Omron CX-Programmer project NewProject (CX-Programmer 9.73)

# PLC NewPLC1: CP2E-N N

## Global symbols (name address type ; comment)
0.00 BOOL  ; PB_EMG
0.01 BOOL  ; Sensor 1m
0.02 BOOL  ; Sensor 1,5 M
0.04 BOOL  ; Sensor Drop
0.06 BOOL  ; Sensor Clean BWD
0.07 BOOL  ; S Home 2
0.08 BOOL  ; S Home 2
0.11 BOOL  ; EMG/PB
100.04 BOOL  ; Q_Break1
100.05 BOOL  ; Q_Break2
100.06 BOOL  ; Q_EN1
100.07 BOOL  ; Q_EN2
101.00 BOOL  ; Cylinder_CLEAN
101.01 BOOL  ; Cylinder_DROP
101.02 BOOL  ; Motor_Down
101.03 BOOL  ; Motor_Up
101.07 BOOL  ; Test Break
200 CHANNEL  ; Timer Clean
280.07 BOOL  ; Ax0 Error
A274 CHANNEL  ; Ax1 Pulse
A276 CHANNEL  ; Ax0 Current PLS
A277 CHANNEL  ; Ax1 Current PLS
A278 CHANNEL  ; Ax1 Pulse Org
A280.04 BOOL  ; Ax0 Busy
A280.05 BOOL  ; Ax0 No Org
A280.06 BOOL  ; Ax0 at Org
A280.07 BOOL  ; Ax0 Error
A281.04 BOOL  ; Ax1 Bussy
A286 CHANNEL  ; Ax1 Current PLS
A540.08 BOOL  ; Ax0 CW-Limit Input
A540.09 BOOL  ; Ax0 CCW-Limit Input
D0 CHANNEL  ; $?St$Bk?_#[4] / Value"0"$?St$Bk?_#[4]
D10 CHANNEL  ; Point A Data
D100 CHANNEL  ; Axo Acceleration
D101 CHANNEL  ; Ax0 Deceleration
D102 CHANNEL  ; Target Frequency
D104 CHANNEL  ; Ax0 Number PLS Output
D105 CHANNEL  ; Ax1 Number PLS Output
D106 CHANNEL  ; Start Frequency
D110 CHANNEL  ; Ax1 Acceleration
D111 CHANNEL  ; Ax1 Deceleration
D112 CHANNEL  ; Target Frequency1
D114 CHANNEL  ; Ax1 Number PLS Output
D116 CHANNEL  ; Start Frequncy1
D12 CHANNEL  ; Point B Data
D120 CHANNEL  ; Ax1 Acceleration
D124 CHANNEL  ; Ax1 Number PLS Output
D126 CHANNEL  ; Start Frequency
D14 CHANNEL  ; Point C Data
D20 CHANNEL  ; Point A2 Data
D22 CHANNEL  ; Point B2 Data
D24 CHANNEL  ; Point C2 Data
D276 CHANNEL  ; Ax0 Current PLS
D277 CHANNEL  ; Ax1 Current PLS
D278 CHANNEL  ; Ax1 PLS
D286 CHANNEL  ; Ax1 Current PLS
T002 BOOL  ; T Clean
T003 BOOL  ; Active DROP
T004 BOOL  ; Active Motor Up
T005 BOOL  ; Timer Continue
T010 BOOL  ; Ax0 Jog High
T011 BOOL  ; Ax1 Jog High
W0.02 BOOL  ; PB Ax0 Org
W0.03 BOOL  ; Axis0 Jog(+)
W0.04 BOOL  ; Axis Jog(-)
W0.05 BOOL  ; PB Ax1 Org
W0.06 BOOL  ; Axis1 Jog(+)
W0.07 BOOL  ; Axis1 Jog(-)
W0.08 BOOL  ; Init Done
W100.00 BOOL  ; No Use
W100.01 BOOL  ; BREAK ACTIVE
W100.02 BOOL  ; ENA 1
W100.03 BOOL  ; INI MOTOR
W100.04 BOOL  ; BREAK 2
W100.07 BOOL  ; ENA 2
W10.00 BOOL  ; Ax0 Recover Org Start
W10.01 BOOL  ; Ax0 Recover Org Start PLS
W10.02 BOOL  ; Ax0 Org Return
W10.03 BOOL  ; Ax0 Org Returning
W10.04 BOOL  ; Ax0 at Org
W10.05 BOOL  ; Init
W10.06 BOOL  ; Ax0 Moving
W10.14 BOOL  ; Ax1 Recover
W10.15 BOOL  ; Ax0 Recover C
W11.00 BOOL  ; 10.01
W11.01 BOOL  ; Ax1 Recover Org Start PLS
W11.10 BOOL  ; Teach A2
W11.11 BOOL  ; Teach B2
W11.12 BOOL  ; Teach C2
W12.00 BOOL  ; Button Home
W12.01 BOOL  ; M_Home 1
W12.02 BOOL  ; Sens Home 1
W12.03 BOOL  ; M_Break 1
W12.04 BOOL  ; M_Break 2
W12.10 BOOL  ; M1_Ready
W12.11 BOOL  ; M2_Ready
W12.12 BOOL  ; Break M1 Deactive
W12.13 BOOL  ; M2_Break Deactive
W13.00 BOOL  ; Button Home2
W13.01 BOOL  ; M_Home 2
W13.02 BOOL  ; Sens_Home2
W14.00 BOOL  ; Teach A2
W14.01 BOOL  ; Teach B2
W14.02 BOOL  ; Teach C2
W15.00 BOOL  ; Point A2 Run
W15.01 BOOL  ; Point B2 Run
W15.02 BOOL  ; Point C2 Run
W15.03 BOOL  ; Home All
W16.00 BOOL  ; IO Clean
W16.01 BOOL  ; IO DROP
W16.02 BOOL  ; M_Mtr_Down
W16.03 BOOL  ; UP 1.5m
W16.04 BOOL  ; Up 1m
W16.05 BOOL  ; FINISH
W16.06 BOOL  ; Go Up
W16.07 BOOL  ; Stop Home
W17.00 BOOL  ; Manual UP
W17.01 BOOL  ; Manual Down
W1.00 BOOL  ; Ax0 Jog High Speed
W1.01 BOOL  ; Ax0 Jog(+)
W1.02 BOOL  ; Ax0 Jog(-)
W1.03 BOOL  ; Ax1 Jog High Speed
W1.04 BOOL  ; Ax1 Jog(+)
W1.05 BOOL  ; Ax1 Jog(-)
W1.08 BOOL  ; Init Done2
W1.10 BOOL  ; Teach Point A
W1.11 BOOL  ; Teah Point B
W1.12 BOOL  ; Teach Point C
W20.00 BOOL  ; No Use
W20.01 BOOL  ; Sens Home
W20.02 BOOL  ; Sens CW
W20.03 BOOL  ; Sens CCW
W2.00 BOOL  ; Point A Run
W2.01 BOOL  ; Point B Run
W2.02 BOOL  ; Point C Run
W2.10 BOOL  ; Point A2 Run
W2.11 BOOL  ; Point B2 Run
W2.12 BOOL  ; Point C2 Run
W3.00 BOOL  ; Point A Proses
W3.01 BOOL  ; Point A Trigger
W3.02 BOOL  ; Ax0 at Point A
W3.10 BOOL  ; Point A2 Proses
W3.11 BOOL  ; Point A2 Trigger
W3.12 BOOL  ; Ax0 at Point A2
W4.00 BOOL  ; Point B Process
W4.01 BOOL  ; Point B Trigger
W4.02 BOOL  ; Ax0 at Point B
W4.10 BOOL  ; Point B2 Progress
W4.11 BOOL  ; Point B2 Trigger
W4.12 BOOL  ; Ax1 at Point B
W5.00 BOOL  ; Point C Progress
W5.01 BOOL  ; Point C Trigger
W5.02 BOOL  ; Ax0 at Point C
W5.10 BOOL  ; Point C2 Progress
W5.11 BOOL  ; Point C2 Trigger
W5.12 BOOL  ; Ax1 at Point C
W6.00 BOOL  ; Sensor Trig
W6.01 BOOL  ; Trig Off
W7.00 BOOL  ; PB_START
W7.01 BOOL  ; M_Start
W7.02 BOOL  ; PB_STOP
W7.03 BOOL  ; PB_HOME
W7.04 BOOL  ; RUN 1or1.5
W7.05 BOOL  ; RUN 1m
W7.06 BOOL  ; PB_Continue
W99.01 BOOL  ; LOCK

## Program NewProgram1 (cyclic task 0)
Local symbols
NOT BOOL

### Section Axis1_Org

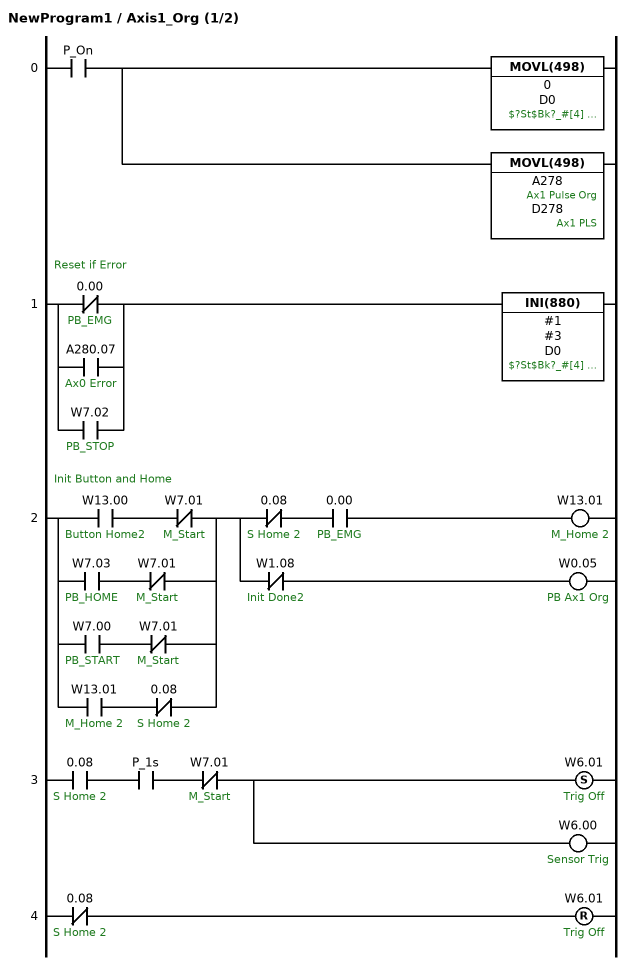
; rung 0
LD P_On
MOVL(498) 0 D0  ; $?St$Bk?_#[4] / Value"0"$?St$Bk?_#[4]
MOVL(498) A278 D278  ; Ax1 Pulse Org, Ax1 PLS
; rung 1: Reset if Error
LDNOT 0.00  ; PB_EMG
OR A280.07  ; Ax0 Error
OR W7.02  ; PB_STOP
INI(880) #1 #3 D0  ; $?St$Bk?_#[4] / Value"0"$?St$Bk?_#[4]
; rung 2: Init Button and Home
LD W13.00  ; Button Home2
ANDNOT W7.01  ; M_Start
LD W7.03  ; PB_HOME
ANDNOT W7.01  ; M_Start
ORLD
LD W7.00  ; PB_START
ANDNOT W7.01  ; M_Start
ORLD
LD W13.01  ; M_Home 2
ANDNOT 0.08  ; S Home 2
ORLD
OUT TR0
ANDNOT 0.08  ; S Home 2
AND 0.00  ; PB_EMG
OUT W13.01  ; M_Home 2
LD TR0
ANDNOT W1.08  ; Init Done2
OUT W0.05  ; PB Ax1 Org
; rung 3
LD 0.08  ; S Home 2
AND P_1s
ANDNOT W7.01  ; M_Start
SET W6.01  ; Trig Off
OUT W6.00  ; Sensor Trig
; rung 4
LDNOT 0.08  ; S Home 2
RSET W6.01  ; Trig Off

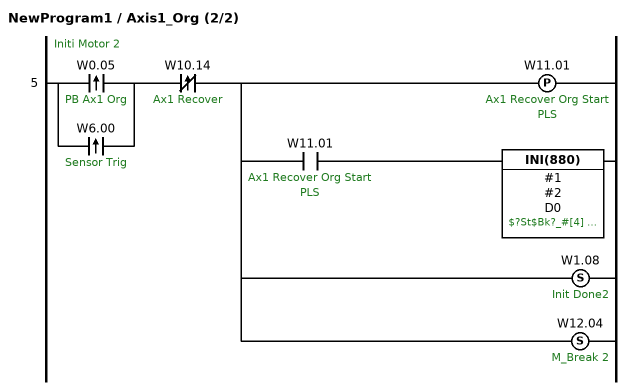
; rung 5: Initi Motor 2
@LD W0.05  ; PB Ax1 Org
@OR W6.00  ; Sensor Trig
@ANDNOT W10.14  ; Ax1 Recover
OUT TR0
DIFU(013) W11.01  ; Ax1 Recover Org Start PLS
AND W11.01  ; Ax1 Recover Org Start PLS
INI(880) #1 #2 D0  ; $?St$Bk?_#[4] / Value"0"$?St$Bk?_#[4]
LD TR0
SET W1.08  ; Init Done2
SET W12.04  ; M_Break 2

### Section Axis1_Jog

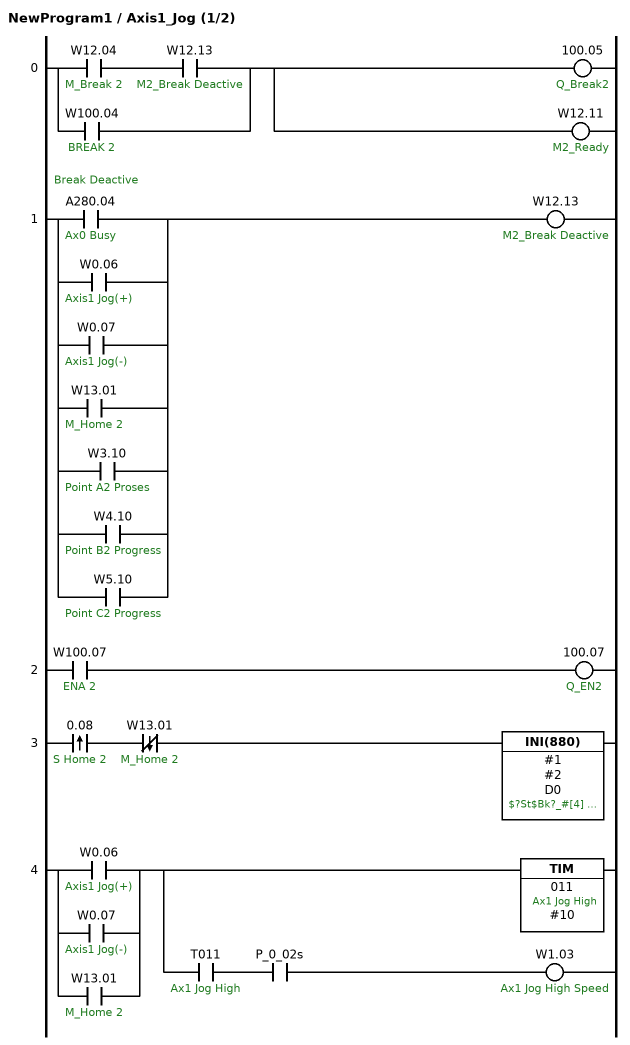
; rung 0
LD W12.04  ; M_Break 2
AND W12.13  ; M2_Break Deactive
OR W100.04  ; BREAK 2
OUT 100.05  ; Q_Break2
OUT W12.11  ; M2_Ready
; rung 1: Break Deactive
LD A280.04  ; Ax0 Busy
OR W0.06  ; Axis1 Jog(+)
OR W0.07  ; Axis1 Jog(-)
OR W13.01  ; M_Home 2
OR W3.10  ; Point A2 Proses
OR W4.10  ; Point B2 Progress
OR W5.10  ; Point C2 Progress
OUT W12.13  ; M2_Break Deactive
; rung 2
LD W100.07  ; ENA 2
OUT 100.07  ; Q_EN2
; rung 3
@LD 0.08  ; S Home 2
%ANDNOT W13.01  ; M_Home 2
INI(880) #1 #2 D0  ; $?St$Bk?_#[4] / Value"0"$?St$Bk?_#[4]
; rung 4
LD W0.06  ; Axis1 Jog(+)
OR W0.07  ; Axis1 Jog(-)
OR W13.01  ; M_Home 2
TIM 011 #10  ; Ax1 Jog High
AND T011  ; Ax1 Jog High
AND P_0_02s
OUT W1.03  ; Ax1 Jog High Speed

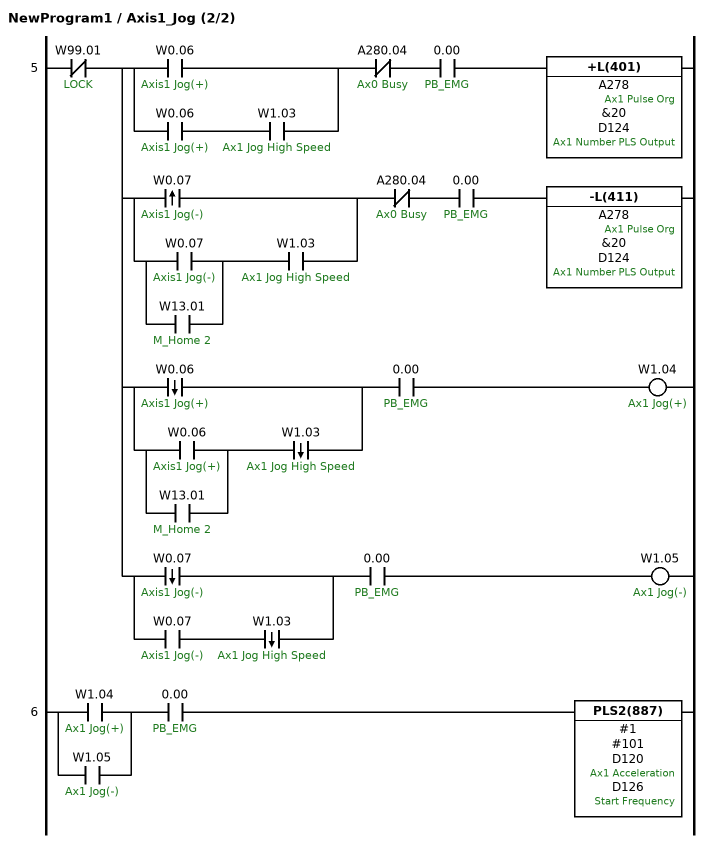
; rung 5
LDNOT W99.01  ; LOCK
OUT TR0
LD W0.06  ; Axis1 Jog(+)
LD W0.06  ; Axis1 Jog(+)
AND W1.03  ; Ax1 Jog High Speed
ORLD
ANDLD
ANDNOT A280.04  ; Ax0 Busy
AND 0.00  ; PB_EMG
+L(401) A278 &20 D124  ; Ax1 Pulse Org, Ax1 Number PLS Output
LD TR0
@LD W0.07  ; Axis1 Jog(-)
LD W0.07  ; Axis1 Jog(-)
OR W13.01  ; M_Home 2
AND W1.03  ; Ax1 Jog High Speed
ORLD
ANDLD
ANDNOT A280.04  ; Ax0 Busy
AND 0.00  ; PB_EMG
-L(411) A278 &20 D124  ; Ax1 Pulse Org, Ax1 Number PLS Output
LD TR0
%LD W0.06  ; Axis1 Jog(+)
LD W0.06  ; Axis1 Jog(+)
OR W13.01  ; M_Home 2
%AND W1.03  ; Ax1 Jog High Speed
ORLD
ANDLD
AND 0.00  ; PB_EMG
OUT W1.04  ; Ax1 Jog(+)
LD TR0
%LD W0.07  ; Axis1 Jog(-)
LD W0.07  ; Axis1 Jog(-)
%AND W1.03  ; Ax1 Jog High Speed
ORLD
ANDLD
AND 0.00  ; PB_EMG
OUT W1.05  ; Ax1 Jog(-)
; rung 6
LD W1.04  ; Ax1 Jog(+)
OR W1.05  ; Ax1 Jog(-)
AND 0.00  ; PB_EMG
PLS2(887) #1 #101 D120 D126  ; Ax1 Acceleration, Start Frequency

### Section Axis1_Point_Run

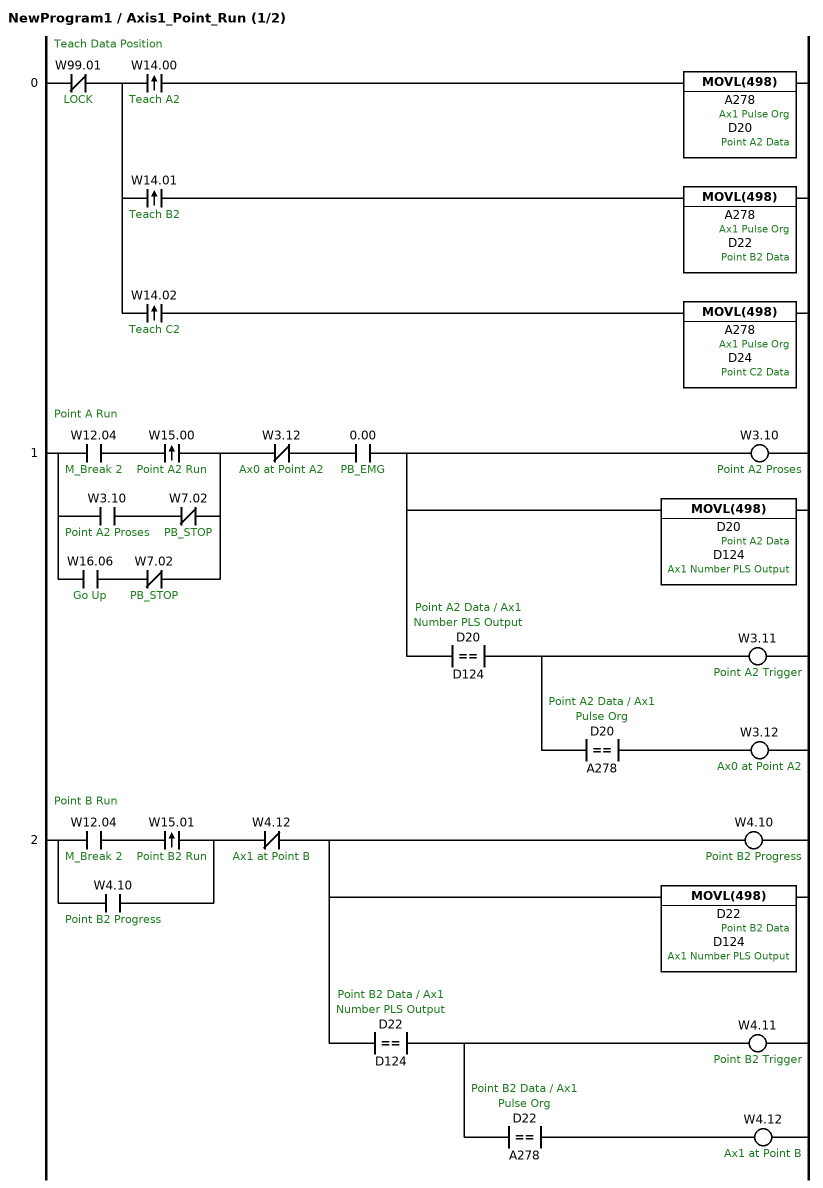
; rung 0: Teach Data Position
LDNOT W99.01  ; LOCK
OUT TR0
@AND W14.00  ; Teach A2
MOVL(498) A278 D20  ; Ax1 Pulse Org, Point A2 Data
LD TR0
@AND W14.01  ; Teach B2
MOVL(498) A278 D22  ; Ax1 Pulse Org, Point B2 Data
LD TR0
@AND W14.02  ; Teach C2
MOVL(498) A278 D24  ; Ax1 Pulse Org, Point C2 Data
; rung 1: Point A Run
LD W12.04  ; M_Break 2
@AND W15.00  ; Point A2 Run
LD W3.10  ; Point A2 Proses
ANDNOT W7.02  ; PB_STOP
ORLD
LD W16.06  ; Go Up
ANDNOT W7.02  ; PB_STOP
ORLD
ANDNOT W3.12  ; Ax0 at Point A2
AND 0.00  ; PB_EMG
OUT W3.10  ; Point A2 Proses
MOVL(498) D20 D124  ; Point A2 Data, Ax1 Number PLS Output
AND=L(301) D20 D124  ; Point A2 Data, Ax1 Number PLS Output
OUT W3.11  ; Point A2 Trigger
AND=L(301) D20 A278  ; Point A2 Data, Ax1 Pulse Org
OUT W3.12  ; Ax0 at Point A2
; rung 2: Point B Run
LD W12.04  ; M_Break 2
@AND W15.01  ; Point B2 Run
OR W4.10  ; Point B2 Progress
ANDNOT W4.12  ; Ax1 at Point B
OUT W4.10  ; Point B2 Progress
MOVL(498) D22 D124  ; Point B2 Data, Ax1 Number PLS Output
AND=L(301) D22 D124  ; Point B2 Data, Ax1 Number PLS Output
OUT W4.11  ; Point B2 Trigger
AND=L(301) D22 A278  ; Point B2 Data, Ax1 Pulse Org
OUT W4.12  ; Ax1 at Point B

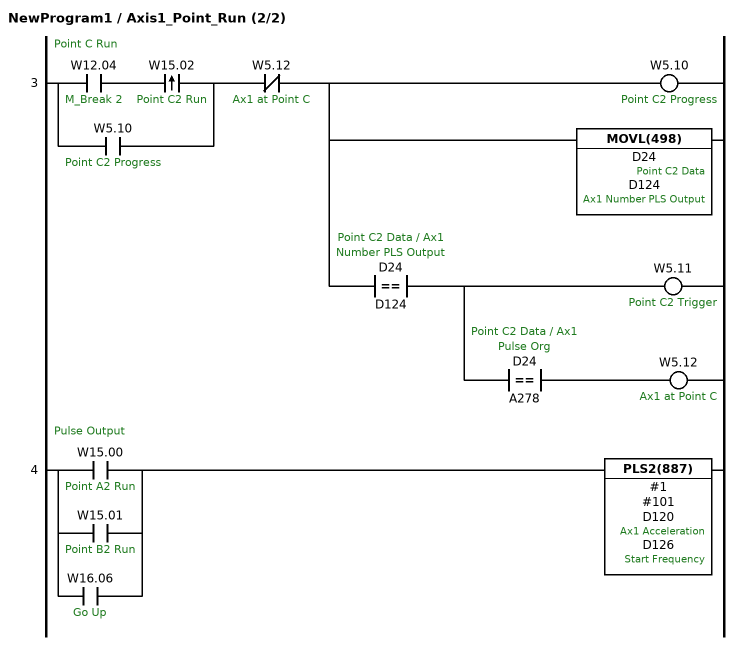
; rung 3: Point C Run
LD W12.04  ; M_Break 2
@AND W15.02  ; Point C2 Run
OR W5.10  ; Point C2 Progress
ANDNOT W5.12  ; Ax1 at Point C
OUT W5.10  ; Point C2 Progress
MOVL(498) D24 D124  ; Point C2 Data, Ax1 Number PLS Output
AND=L(301) D24 D124  ; Point C2 Data, Ax1 Number PLS Output
OUT W5.11  ; Point C2 Trigger
AND=L(301) D24 A278  ; Point C2 Data, Ax1 Pulse Org
OUT W5.12  ; Ax1 at Point C
; rung 4: Pulse Output
LD W15.00  ; Point A2 Run
OR W15.01  ; Point B2 Run
OR W16.06  ; Go Up
PLS2(887) #1 #101 D120 D126  ; Ax1 Acceleration, Start Frequency

### Section MOTOR_DROP_TEST

### Section Program

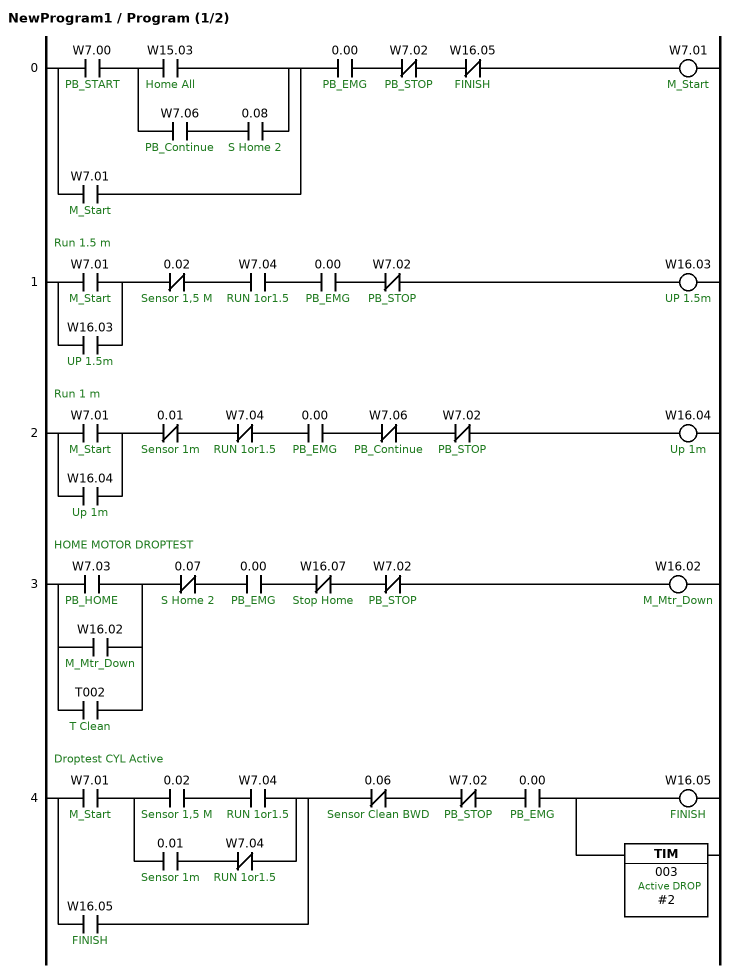
; rung 0
LD W7.00  ; PB_START
LD W15.03  ; Home All
LD W7.06  ; PB_Continue
AND 0.08  ; S Home 2
ORLD
ANDLD
OR W7.01  ; M_Start
AND 0.00  ; PB_EMG
ANDNOT W7.02  ; PB_STOP
ANDNOT W16.05  ; FINISH
OUT W7.01  ; M_Start
; rung 1: Run 1.5 m
LD W7.01  ; M_Start
OR W16.03  ; UP 1.5m
ANDNOT 0.02  ; Sensor 1,5 M
AND W7.04  ; RUN 1or1.5
AND 0.00  ; PB_EMG
ANDNOT W7.02  ; PB_STOP
OUT W16.03  ; UP 1.5m
; rung 2: Run 1 m
LD W7.01  ; M_Start
OR W16.04  ; Up 1m
ANDNOT 0.01  ; Sensor 1m
ANDNOT W7.04  ; RUN 1or1.5
AND 0.00  ; PB_EMG
ANDNOT W7.06  ; PB_Continue
ANDNOT W7.02  ; PB_STOP
OUT W16.04  ; Up 1m
; rung 3: HOME MOTOR DROPTEST
LD W7.03  ; PB_HOME
OR W16.02  ; M_Mtr_Down
OR T002  ; T Clean
ANDNOT 0.07  ; S Home 2
AND 0.00  ; PB_EMG
ANDNOT W16.07  ; Stop Home
ANDNOT W7.02  ; PB_STOP
OUT W16.02  ; M_Mtr_Down
; rung 4: Droptest CYL Active
LD W7.01  ; M_Start
LD 0.02  ; Sensor 1,5 M
AND W7.04  ; RUN 1or1.5
LD 0.01  ; Sensor 1m
ANDNOT W7.04  ; RUN 1or1.5
ORLD
ANDLD
OR W16.05  ; FINISH
ANDNOT 0.06  ; Sensor Clean BWD
ANDNOT W7.02  ; PB_STOP
AND 0.00  ; PB_EMG
OUT W16.05  ; FINISH
TIM 003 #2  ; Active DROP

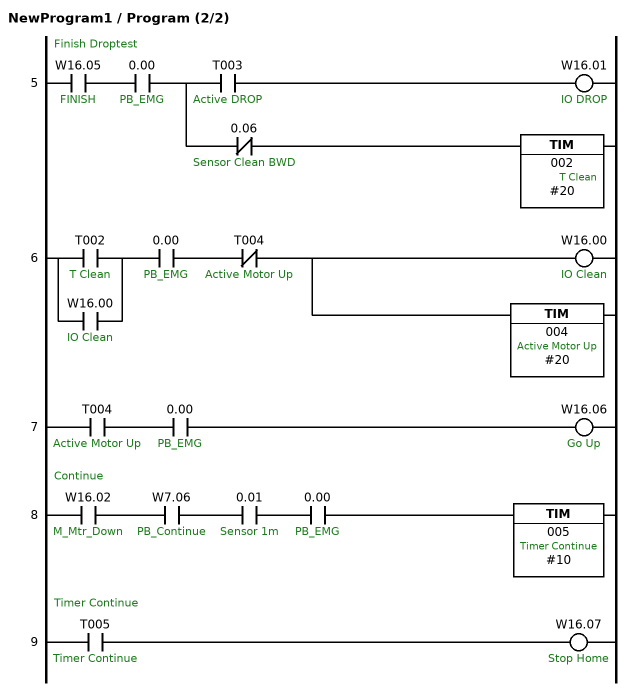
; rung 5: Finish Droptest
LD W16.05  ; FINISH
AND 0.00  ; PB_EMG
OUT TR0
AND T003  ; Active DROP
OUT W16.01  ; IO DROP
LD TR0
ANDNOT 0.06  ; Sensor Clean BWD
TIM 002 #20  ; T Clean
; rung 6
LD T002  ; T Clean
OR W16.00  ; IO Clean
AND 0.00  ; PB_EMG
ANDNOT T004  ; Active Motor Up
OUT W16.00  ; IO Clean
TIM 004 #20  ; Active Motor Up
; rung 7
LD T004  ; Active Motor Up
AND 0.00  ; PB_EMG
OUT W16.06  ; Go Up
; rung 8: Continue
LD W16.02  ; M_Mtr_Down
AND W7.06  ; PB_Continue
AND 0.01  ; Sensor 1m
AND 0.00  ; PB_EMG
TIM 005 #10  ; Timer Continue
; rung 9: Timer Continue
LD T005  ; Timer Continue
OUT W16.07  ; Stop Home

### Section I_O

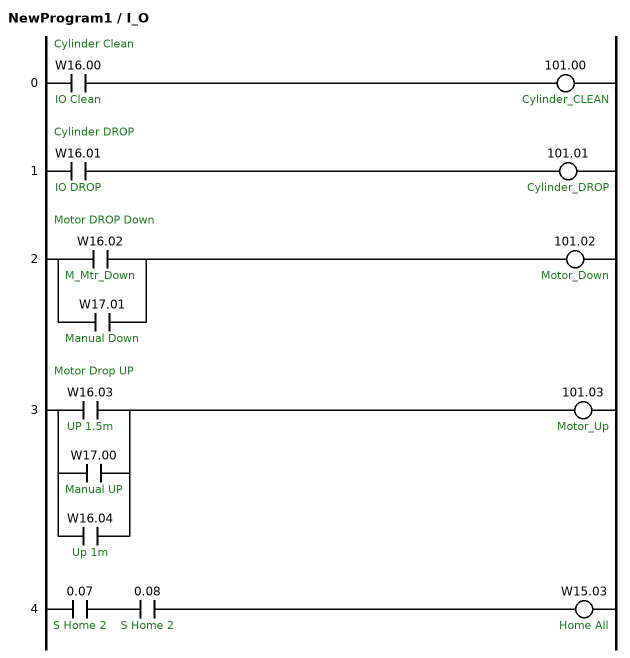
; rung 0: Cylinder Clean
LD W16.00  ; IO Clean
OUT 101.00  ; Cylinder_CLEAN
; rung 1: Cylinder DROP
LD W16.01  ; IO DROP
OUT 101.01  ; Cylinder_DROP
; rung 2: Motor DROP Down
LD W16.02  ; M_Mtr_Down
OR W17.01  ; Manual Down
OUT 101.02  ; Motor_Down
; rung 3: Motor Drop UP
LD W16.03  ; UP 1.5m
OR W17.00  ; Manual UP
OR W16.04  ; Up 1m
OUT 101.03  ; Motor_Up
; rung 4
LD 0.07  ; S Home 2
AND 0.08  ; S Home 2
OUT W15.03  ; Home All

### Section END
; rung 0
END(001)